FUNCTION_BLOCK E_RESTART (* Service Interface Function Block Type *)
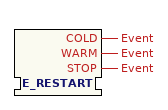
  EVENT_OUTPUT
    COLD; (* Information on cold restart *)
    WARM; (* Information on warm restart *)
    STOP; (* information that the resource is to be stopped *)
  END_EVENT
  SERVICE E_RESTART/RESOURCE (* Service Interface Function Block Type *)
    SEQUENCE cold_restart
      RESOURCE.start() -> E_RESTART.START();
    END_SEQUENCE
    SEQUENCE warm_restart
      RESOURCE.restart() -> E_RESTART.WARM();
    END_SEQUENCE
    SEQUENCE stopping
      RESOURCE.stop() -> E_RESTART.STOP();
    END_SEQUENCE
  END_SERVICE
END_FUNCTION_BLOCK
